  MoveL 717 to (-24.58, 53.5, 24) mm, rotated rx -180 ry 0 rz 180 deg; joints [-1.626, -7.129, -30.226, -175.862, -23.152, -3.806]
  MoveL 718 to (-28.76, 51.39, 24) mm, rotated rx 180 ry 0 rz 180 deg; joints [-1.72, -7.341, -30.414, -175.619, -23.133, -4.03]
  MoveL 719 to (-33.23, 48.62, 24) mm, rotated rx -180 ry 0 rz -180 deg; joints [-1.842, -7.567, -30.613, -175.303, -23.115, -4.321]
  MoveL 720 to (-37.7, 45.24, 24) mm, rotated rx 180 ry 0 rz 180 deg; joints [-1.991, -7.792, -30.809, -174.919, -23.098, -4.675]
  MoveL 721 to (-42.11, 41.08, 24) mm, rotated rx 180 ry 0 rz 180 deg; joints [-2.174, -8.013, -31.001, -174.448, -23.085, -5.11]
  MoveL 722 to (-46.58, 36.05, 24) mm, rotated rx -180 ry 0 rz -180 deg; joints [-2.395, -8.233, -31.193, -173.879, -23.077, -5.634]
  MoveL 723 to (-48.92, 32.78, 24) mm, rotated rx -180 ry 0 rz -180 deg; joints [-2.539, -8.348, -31.291, -173.511, -23.076, -5.974]
  MoveL 724 to (-51.1, 29.15, 24) mm, rotated rx 180 ry 0 rz 180 deg; joints [-2.698, -8.452, -31.382, -173.104, -23.079, -6.349]
  MoveL 725 to (-52.53, 26.41, 24) mm, rotated rx -180 ry 0 rz 180 deg; joints [-2.818, -8.519, -31.439, -172.797, -23.083, -6.631]
  MoveL 726 to (-54.51, 22.28, 24) mm, rotated rx 180 ry 0 rz 180 deg; joints [-2.998, -8.611, -31.519, -172.336, -23.092, -7.056]
  MoveL 727 to (-56.61, 15.99, 24) mm, rotated rx -180 ry 0 rz 180 deg; joints [-3.272, -8.702, -31.597, -171.64, -23.115, -7.697]
  MoveL 728 to (-57.94, 10.54, 24) mm, rotated rx -180 ry 0 rz 180 deg; joints [-3.509, -8.755, -31.642, -171.04, -23.14, -8.249]
  MoveL 729 to (-58.64, 4.96, 24) mm, rotated rx 180 ry 0 rz 180 deg; joints [-3.75, -8.773, -31.657, -170.433, -23.173, -8.807]
  MoveL 730 to (-58.87, 0.71, 24) mm, rotated rx 180 ry 0 rz 180 deg; joints [-3.932, -8.77, -31.655, -169.976, -23.202, -9.228]
  MoveL 731 to (-58.77, -3.71, 24) mm, rotated rx 180 ry 0 rz 180 deg; joints [-4.121, -8.748, -31.636, -169.505, -23.236, -9.661]
  MoveL 732 to (-58.13, -9.36, 24) mm, rotated rx -180 ry 0 rz -180 deg; joints [-4.361, -8.694, -31.589, -168.91, -23.285, -10.206]
  MoveL 733 to (-56.57, -16.2, 24) mm, rotated rx -180 ry 0 rz 180 deg; joints [-4.648, -8.585, -31.496, -168.205, -23.353, -10.853]
  MoveL 734 to (-54.78, -21.48, 24) mm, rotated rx -180 ry 0 rz -180 deg; joints [-4.866, -8.469, -31.397, -167.673, -23.41, -11.34]
  MoveL 735 to (-52.18, -27.29, 24) mm, rotated rx -180 ry 0 rz 180 deg; joints [-5.103, -8.309, -31.258, -167.099, -23.48, -11.864]
  MoveL 736 to (-50.38, -30.48, 24) mm, rotated rx -180 ry 0 rz 180 deg; joints [-5.232, -8.201, -31.164, -166.792, -23.521, -12.145]
  MoveL 737 to (-46.66, -35.77, 24) mm, rotated rx -180 ry 0 rz 180 deg; joints [-5.441, -7.983, -30.976, -166.296, -23.593, -12.596]
  MoveL 738 to (-43.36, -39.85, 24) mm, rotated rx -180 ry 0 rz 180 deg; joints [-5.599, -7.793, -30.81, -165.924, -23.652, -12.935]
  MoveL 739 to (-39.52, -43.58, 24) mm, rotated rx -180 ry 0 rz 180 deg; joints [-5.74, -7.577, -30.621, -165.597, -23.71, -13.232]
  MoveL 740 to (-36.23, -46.33, 24) mm, rotated rx -180 ry 0 rz -180 deg; joints [-5.842, -7.393, -30.46, -165.365, -23.755, -13.442]
  Set speed (16.7 mm/s)
  MoveL 741 to (-35.66, -46.6, 24) mm, rotated rx 180 ry 0 rz 180 deg; joints [-5.85, -7.363, -30.433, -165.347, -23.761, -13.458]
  MoveL 742 to (-35.05, -46.54, 24) mm, rotated rx -180 ry 0 rz -180 deg; joints [-5.845, -7.331, -30.405, -165.361, -23.763, -13.445]
  MoveL 743 to (-34.54, -46.18, 24) mm, rotated rx 180 ry 0 rz 180 deg; joints [-5.828, -7.307, -30.384, -165.404, -23.762, -13.405]
  MoveL 744 to (-34.69, -44.49, 24) mm, rotated rx -180 ry 0 rz 180 deg; joints [-5.758, -7.324, -30.399, -165.572, -23.744, -13.252]
  Set speed (1000.0 mm/s)
  MoveL 745 to (-26.21, -33.57, 24) mm, rotated rx -180 ry 0 rz -180 deg; joints [-5.268, -6.943, -30.062, -166.784, -23.68, -12.137]
  Set speed (5.0 mm/s)
  MoveL 746 to (-26.21, -33.57, 18) mm, rotated rx -180 ry 0 rz 180 deg; joints [-5.268, -6.879, -30.286, -166.933, -23.96, -11.975]
  MoveL 747 to (-27.9, -33.77, 18) mm, rotated rx 180 ry 0 rz 180 deg; joints [-5.283, -6.964, -30.362, -166.892, -23.954, -12.014]
  MoveL 748 to (-28.14, -34.34, 18) mm, rotated rx -180 ry 0 rz 180 deg; joints [-5.308, -6.974, -30.371, -166.831, -23.958, -12.069]
  MoveL 749 to (-28.07, -34.96, 18) mm, rotated rx 180 ry 0 rz 180 deg; joints [-5.333, -6.967, -30.365, -166.771, -23.964, -12.124]
  MoveL 750 to (-27.69, -35.46, 18) mm, rotated rx 180 ry 0 rz 180 deg; joints [-5.353, -6.946, -30.345, -166.726, -23.97, -12.165]
  Set speed (16.7 mm/s)
  MoveL 751 to (-26.15, -36.67, 18) mm, rotated rx -180 ry 0 rz -180 deg; joints [-5.397, -6.861, -30.27, -166.624, -23.989, -12.257]
  MoveL 752 to (-23.6, -38.37, 18) mm, rotated rx -180 ry 0 rz -180 deg; joints [-5.458, -6.722, -30.147, -166.486, -24.017, -12.382]
  MoveL 753 to (-18.39, -41.25, 18) mm, rotated rx 180 ry 0 rz 180 deg; joints [-5.556, -6.441, -29.896, -166.266, -24.068, -12.579]
  MoveL 754 to (-14.04, -42.78, 18) mm, rotated rx 180 ry 0 rz -180 deg; joints [-5.602, -6.212, -29.69, -166.17, -24.101, -12.665]
  MoveL 755 to (-7.62, -44.52, 18) mm, rotated rx -180 ry 0 rz -180 deg; joints [-5.647, -5.875, -29.387, -166.079, -24.143, -12.745]
  MoveL 756 to (-0.08, -45.16, 18) mm, rotated rx 180 ry 0 rz 180 deg; joints [-5.643, -5.488, -29.036, -166.108, -24.177, -12.714]
  MoveL 757 to (4.54, -44.87, 18) mm, rotated rx 180 ry 0 rz 180 deg; joints [-5.613, -5.255, -28.823, -166.192, -24.191, -12.636]
  MoveL 758 to (10.55, -43.81, 18) mm, rotated rx 180 ry 0 rz 180 deg; joints [-5.546, -4.955, -28.549, -166.365, -24.2, -12.476]
  MoveL 759 to (15.67, -42.36, 18) mm, rotated rx -180 ry 0 rz 180 deg; joints [-5.467, -4.702, -28.316, -166.562, -24.203, -12.294]
  MoveL 760 to (22.77, -38.96, 18) mm, rotated rx -180 ry 0 rz -180 deg; joints [-5.303, -4.359, -27.998, -166.966, -24.193, -11.923]
  MoveL 761 to (23.75, -38.19, 18) mm, rotated rx 180 ry 0 rz 180 deg; joints [-5.269, -4.313, -27.956, -167.05, -24.19, -11.847]
  MoveL 762 to (24.79, -37.75, 18) mm, rotated rx 180 ry 0 rz 180 deg; joints [-5.247, -4.263, -27.909, -167.103, -24.189, -11.798]
  MoveL 763 to (25.87, -36.99, 18) mm, rotated rx -180 ry 0 rz -180 deg; joints [-5.213, -4.212, -27.861, -167.187, -24.185, -11.721]
  MoveL 764 to (31.61, -32.27, 18) mm, rotated rx -180 ry 0 rz -180 deg; joints [-5.003, -3.943, -27.611, -167.697, -24.161, -11.254]
  MoveL 765 to (34.13, -29.42, 18) mm, rotated rx -180 ry 0 rz -180 deg; joints [-4.881, -3.828, -27.503, -167.994, -24.144, -10.982]
  MoveL 766 to (38.38, -23.8, 18) mm, rotated rx -180 ry 0 rz 180 deg; joints [-4.643, -3.637, -27.324, -168.572, -24.112, -10.454]
  MoveL 767 to (40.34, -20.05, 18) mm, rotated rx 180 ry 0 rz 180 deg; joints [-4.487, -3.554, -27.245, -168.948, -24.089, -10.11]
  MoveL 768 to (42.9, -14.11, 18) mm, rotated rx 180 ry 0 rz 180 deg; joints [-4.243, -3.447, -27.145, -169.54, -24.053, -9.569]
  MoveL 769 to (43.73, -10.9, 18) mm, rotated rx -180 ry 0 rz 180 deg; joints [-4.114, -3.417, -27.117, -169.855, -24.033, -9.281]
  MoveL 770 to (45.05, -3.17, 18) mm, rotated rx 180 ry 0 rz 180 deg; joints [-3.803, -3.378, -27.079, -170.611, -23.987, -8.591]
  MoveL 771 to (45.17, 0.09, 18) mm, rotated rx 180 ry 0 rz 180 deg; joints [-3.673, -3.383, -27.084, -170.927, -23.968, -8.302]
  MoveL 772 to (44.61, 6.42, 18) mm, rotated rx -180 ry 0 rz 180 deg; joints [-3.423, -3.431, -27.129, -171.536, -23.93, -7.745]
  MoveL 773 to (43.15, 13.22, 18) mm, rotated rx -180 ry 0 rz 180 deg; joints [-3.156, -3.524, -27.217, -172.188, -23.89, -7.15]
  MoveL 774 to (41.73, 17.09, 18) mm, rotated rx 180 ry 0 rz 180 deg; joints [-3.004, -3.606, -27.295, -172.557, -23.867, -6.813]
  MoveL 775 to (38.05, 24.34, 18) mm, rotated rx -180 ry 0 rz -180 deg; joints [-2.722, -3.811, -27.487, -173.248, -23.823, -6.181]
  MoveL 776 to (34.85, 28.44, 18) mm, rotated rx -180 ry 0 rz 180 deg; joints [-2.564, -3.982, -27.647, -173.635, -23.796, -5.828]
  MoveL 777 to (30.87, 32.97, 18) mm, rotated rx 180 ry 0 rz 180 deg; joints [-2.389, -4.194, -27.845, -174.064, -23.764, -5.436]
  MoveL 778 to (24.7, 37.75, 18) mm, rotated rx -180 ry 0 rz -180 deg; joints [-2.206, -4.517, -28.145, -174.51, -23.725, -5.028]
  MoveL 779 to (24.15, 37.96, 18) mm, rotated rx 180 ry 0 rz 180 deg; joints [-2.198, -4.545, -28.171, -174.528, -23.722, -5.012]
  MoveL 780 to (23.56, 38.41, 18) mm, rotated rx -180 ry 0 rz 180 deg; joints [-2.181, -4.576, -28.2, -174.571, -23.718, -4.973]
  MoveL 781 to (18.35, 41.27, 18) mm, rotated rx 180 ry 0 rz 180 deg; joints [-2.073, -4.846, -28.449, -174.834, -23.688, -4.733]
  MoveL 782 to (14.11, 42.76, 18) mm, rotated rx -180 ry 0 rz 180 deg; joints [-2.019, -5.065, -28.65, -174.965, -23.666, -4.613]
  MoveL 783 to (7.59, 44.53, 18) mm, rotated rx 180 ry 0 rz 180 deg; joints [-1.956, -5.401, -28.957, -175.116, -23.632, -4.476]
  MoveL 784 to (0.04, 45.16, 18) mm, rotated rx 180 ry 0 rz 180 deg; joints [-1.94, -5.787, -29.308, -175.148, -23.596, -4.448]
  MoveL 785 to (-5.87, 44.7, 18) mm, rotated rx 180 ry 0 rz 180 deg; joints [-1.968, -6.089, -29.58, -175.074, -23.569, -4.517]
  MoveL 786 to (-12.92, 43.24, 18) mm, rotated rx -180 ry 0 rz 180 deg; joints [-2.038, -6.448, -29.902, -174.89, -23.538, -4.687]
  MoveL 787 to (-16.08, 42.17, 18) mm, rotated rx 180 ry 0 rz 180 deg; joints [-2.087, -6.609, -30.046, -174.764, -23.525, -4.803]
  MoveL 788 to (-22.99, 38.84, 18) mm, rotated rx 180 ry 0 rz 180 deg; joints [-2.237, -6.957, -30.356, -174.382, -23.499, -5.155]
  MoveL 789 to (-23.69, 38.24, 18) mm, rotated rx 180 ry 0 rz 180 deg; joints [-2.263, -6.992, -30.387, -174.315, -23.497, -5.216]
  MoveL 790 to (-24.82, 37.73, 18) mm, rotated rx -180 ry 0 rz 180 deg; joints [-2.287, -7.049, -30.437, -174.256, -23.493, -5.271]
  MoveL 791 to (-25.9, 36.97, 18) mm, rotated rx 180 ry 0 rz 180 deg; joints [-2.32, -7.103, -30.485, -174.17, -23.49, -5.35]
  MoveL 792 to (-31.55, 32.32, 18) mm, rotated rx 180 ry 0 rz 180 deg; joints [-2.526, -7.385, -30.733, -173.649, -23.477, -5.829]
  MoveL 793 to (-34.16, 29.39, 18) mm, rotated rx 180 ry 0 rz 180 deg; joints [-2.654, -7.512, -30.845, -173.325, -23.475, -6.127]
  MoveL 794 to (-38.41, 23.76, 18) mm, rotated rx -180 ry 0 rz 180 deg; joints [-2.9, -7.718, -31.025, -172.703, -23.477, -6.698]
  MoveL 795 to (-40.36, 20, 18) mm, rotated rx -180 ry 0 rz 180 deg; joints [-3.063, -7.809, -31.104, -172.294, -23.485, -7.075]
  MoveL 796 to (-42.93, 14.05, 18) mm, rotated rx -180 ry 0 rz 180 deg; joints [-3.321, -7.924, -31.205, -171.647, -23.503, -7.669]
  MoveL 797 to (-43.76, 10.82, 18) mm, rotated rx -180 ry 0 rz -180 deg; joints [-3.46, -7.957, -31.233, -171.301, -23.518, -7.986]
  MoveL 798 to (-45.03, 3.4, 18) mm, rotated rx -180 ry 0 rz -180 deg; joints [-3.778, -7.999, -31.27, -170.511, -23.559, -8.711]
  MoveL 799 to (-45.16, 0.22, 18) mm, rotated rx -180 ry 0 rz -180 deg; joints [-3.913, -7.994, -31.266, -170.178, -23.58, -9.016]
  MoveL 800 to (-44.82, -4.92, 18) mm, rotated rx -180 ry 0 rz 180 deg; joints [-4.13, -7.958, -31.234, -169.645, -23.62, -9.504]
  MoveL 801 to (-43.65, -11.27, 18) mm, rotated rx 180 ry 0 rz 180 deg; joints [-4.395, -7.873, -31.16, -168.999, -23.676, -10.095]
  MoveL 802 to (-42.96, -13.88, 18) mm, rotated rx 180 ry 0 rz 180 deg; joints [-4.503, -7.827, -31.12, -168.737, -23.701, -10.334]
  MoveL 803 to (-41.79, -16.95, 18) mm, rotated rx -180 ry 0 rz -180 deg; joints [-4.629, -7.754, -31.056, -168.434, -23.733, -10.611]
  MoveL 804 to (-38.1, -24.27, 18) mm, rotated rx 180 ry 0 rz 180 deg; joints [-4.924, -7.532, -30.862, -167.728, -23.816, -11.255]
  MoveL 805 to (-36.06, -27.07, 18) mm, rotated rx 180 ry 0 rz 180 deg; joints [-5.034, -7.415, -30.759, -167.468, -23.851, -11.491]
  MoveL 806 to (-30.91, -32.94, 18) mm, rotated rx 180 ry 0 rz 180 deg; joints [-5.26, -7.123, -30.502, -166.939, -23.931, -11.972]
  MoveL 807 to (-27.69, -35.46, 18) mm, rotated rx 180 ry 0 rz 180 deg; joints [-5.353, -6.946, -30.345, -166.726, -23.97, -12.165]
  Set speed (16.7 mm/s)
  MoveL 808 to (-27.12, -35.7, 18) mm, rotated rx 180 ry 0 rz 180 deg; joints [-5.361, -6.915, -30.318, -166.708, -23.976, -12.181]
  MoveL 809 to (-26.51, -35.63, 18) mm, rotated rx -180 ry 0 rz -180 deg; joints [-5.355, -6.884, -30.291, -166.723, -23.978, -12.167]
  MoveL 810 to (-26.01, -35.25, 18) mm, rotated rx -180 ry 0 rz -180 deg; joints [-5.338, -6.86, -30.27, -166.767, -23.977, -12.127]
  MoveL 811 to (-26.21, -33.57, 18) mm, rotated rx 180 ry 0 rz 180 deg; joints [-5.268, -6.879, -30.286, -166.933, -23.96, -11.975]
  Set speed (1000.0 mm/s)
  MoveL 812 to (-12.43, -16.45, 18) mm, rotated rx -180 ry 0 rz 180 deg; joints [-4.51, -6.248, -29.723, -168.8, -23.88, -10.262]
  Set speed (5.0 mm/s)
  MoveL 813 to (-12.43, -16.45, 12) mm, rotated rx -180 ry 0 rz -180 deg; joints [-4.51, -6.182, -29.945, -168.925, -24.163, -10.125]
  MoveL 814 to (-14.12, -16.64, 12) mm, rotated rx 180 ry 0 rz 180 deg; joints [-4.523, -6.268, -30.022, -168.89, -24.156, -10.158]
  MoveL 815 to (-14.37, -17.21, 12) mm, rotated rx -180 ry 0 rz -180 deg; joints [-4.547, -6.278, -30.031, -168.831, -24.16, -10.212]
  MoveL 816 to (-14.3, -17.82, 12) mm, rotated rx -180 ry 0 rz -180 deg; joints [-4.572, -6.272, -30.026, -168.77, -24.165, -10.268]
  MoveL 817 to (-13.93, -18.33, 12) mm, rotated rx -180 ry 0 rz -180 deg; joints [-4.592, -6.251, -30.007, -168.724, -24.17, -10.309]
  Set speed (16.7 mm/s)
  MoveL 818 to (-13.27, -18.86, 12) mm, rotated rx 180 ry 0 rz 180 deg; joints [-4.612, -6.215, -29.975, -168.678, -24.178, -10.351]
  MoveL 819 to (-10.86, -20.34, 12) mm, rotated rx 180 ry 0 rz 180 deg; joints [-4.665, -6.086, -29.858, -168.557, -24.2, -10.461]
  MoveL 820 to (-8.3, -21.51, 12) mm, rotated rx -180 ry 0 rz -180 deg; joints [-4.705, -5.95, -29.736, -168.467, -24.22, -10.541]
  MoveL 821 to (-5.71, -22.36, 12) mm, rotated rx -180 ry 0 rz 180 deg; joints [-4.731, -5.814, -29.613, -168.411, -24.238, -10.592]
  MoveL 822 to (-2.84, -23, 12) mm, rotated rx 180 ry 0 rz 180 deg; joints [-4.747, -5.665, -29.479, -168.378, -24.255, -10.621]
  MoveL 823 to (0.04, -23.2, 12) mm, rotated rx 180 ry 0 rz 180 deg; joints [-4.745, -5.518, -29.344, -168.388, -24.268, -10.611]
  MoveL 824 to (2.55, -23.04, 12) mm, rotated rx 180 ry 0 rz 180 deg; joints [-4.73, -5.39, -29.228, -168.429, -24.276, -10.572]
  MoveL 825 to (4.71, -22.63, 12) mm, rotated rx -180 ry 0 rz 180 deg; joints [-4.707, -5.282, -29.129, -168.49, -24.281, -10.516]
  MoveL 826 to (7.7, -21.73, 12) mm, rotated rx -180 ry 0 rz 180 deg; joints [-4.66, -5.134, -28.994, -168.607, -24.285, -10.408]
  MoveL 827 to (10.34, -20.61, 12) mm, rotated rx 180 ry 0 rz 180 deg; joints [-4.606, -5.004, -28.875, -168.742, -24.286, -10.284]
  MoveL 828 to (12.82, -19.16, 12) mm, rotated rx -180 ry 0 rz 180 deg; joints [-4.539, -4.884, -28.765, -168.906, -24.283, -10.134]
  MoveL 829 to (15.05, -17.47, 12) mm, rotated rx 180 ry 0 rz 180 deg; joints [-4.463, -4.778, -28.667, -169.09, -24.278, -9.965]
  MoveL 830 to (17.03, -15.54, 12) mm, rotated rx -180 ry 0 rz 180 deg; joints [-4.379, -4.684, -28.581, -169.296, -24.271, -9.777]
  MoveL 831 to (18.85, -13.28, 12) mm, rotated rx 180 ry 0 rz 180 deg; joints [-4.282, -4.601, -28.504, -169.531, -24.261, -9.562]
  MoveL 832 to (20.34, -10.86, 12) mm, rotated rx 180 ry 0 rz 180 deg; joints [-4.18, -4.534, -28.442, -169.778, -24.249, -9.337]
  MoveL 833 to (21.5, -8.33, 12) mm, rotated rx -180 ry 0 rz -180 deg; joints [-4.074, -4.485, -28.396, -170.033, -24.236, -9.104]
  MoveL 834 to (22.34, -5.7, 12) mm, rotated rx -180 ry 0 rz -180 deg; joints [-3.966, -4.452, -28.366, -170.295, -24.221, -8.865]
  MoveL 835 to (22.85, -2.99, 12) mm, rotated rx -180 ry 0 rz -180 deg; joints [-3.855, -4.435, -28.35, -170.562, -24.206, -8.621]
  MoveL 836 to (23.04, 0.44, 12) mm, rotated rx -180 ry 0 rz 180 deg; joints [-3.716, -4.437, -28.352, -170.897, -24.185, -8.315]
  MoveL 837 to (22.58, 4.55, 12) mm, rotated rx -180 ry 0 rz -180 deg; joints [-3.551, -4.474, -28.386, -171.295, -24.159, -7.953]
  MoveL 838 to (21.92, 7.05, 12) mm, rotated rx 180 ry 0 rz 180 deg; joints [-3.452, -4.515, -28.424, -171.534, -24.143, -7.735]
  MoveL 839 to (20.59, 10.37, 12) mm, rotated rx 180 ry 0 rz 180 deg; joints [-3.321, -4.592, -28.496, -171.85, -24.12, -7.447]
  MoveL 840 to (19.25, 12.68, 12) mm, rotated rx 180 ry 0 rz -180 deg; joints [-3.231, -4.667, -28.565, -172.067, -24.102, -7.249]
  MoveL 841 to (17.5, 15.01, 12) mm, rotated rx -180 ry 0 rz -180 deg; joints [-3.14, -4.763, -28.653, -172.286, -24.084, -7.05]
  MoveL 842 to (15.49, 17.08, 12) mm, rotated rx 180 ry 0 rz 180 deg; joints [-3.061, -4.871, -28.752, -172.476, -24.066, -6.876]
  MoveL 843 to (13.35, 18.8, 12) mm, rotated rx 180 ry 0 rz 180 deg; joints [-2.995, -4.984, -28.857, -172.633, -24.049, -6.734]
  MoveL 844 to (10.93, 20.3, 12) mm, rotated rx -180 ry 0 rz -180 deg; joints [-2.939, -5.111, -28.973, -172.766, -24.032, -6.612]
  MoveL 845 to (8.27, 21.52, 12) mm, rotated rx 180 ry 0 rz 180 deg; joints [-2.895, -5.25, -29.101, -172.872, -24.015, -6.517]
  MoveL 846 to (5.67, 22.37, 12) mm, rotated rx 180 ry 0 rz 180 deg; joints [-2.866, -5.385, -29.224, -172.94, -24, -6.455]
  MoveL 847 to (2.81, 23, 12) mm, rotated rx 180 ry 0 rz 180 deg; joints [-2.846, -5.533, -29.358, -172.985, -23.985, -6.415]
  MoveL 848 to (0.03, 23.2, 12) mm, rotated rx -180 ry 0 rz 180 deg; joints [-2.843, -5.675, -29.488, -172.987, -23.972, -6.413]
  MoveL 849 to (-2.49, 23.04, 12) mm, rotated rx 180 ry 0 rz 180 deg; joints [-2.855, -5.803, -29.604, -172.956, -23.961, -6.443]
  MoveL 850 to (-4.65, 22.65, 12) mm, rotated rx -180 ry 0 rz 180 deg; joints [-2.876, -5.913, -29.703, -172.902, -23.953, -6.492]
  MoveL 851 to (-7.73, 21.72, 12) mm, rotated rx -180 ry 0 rz 180 deg; joints [-2.92, -6.069, -29.843, -172.789, -23.943, -6.597]
  MoveL 852 to (-10.37, 20.59, 12) mm, rotated rx -180 ry 0 rz -180 deg; joints [-2.972, -6.201, -29.962, -172.657, -23.936, -6.718]
  MoveL 853 to (-12.76, 19.2, 12) mm, rotated rx 180 ry 0 rz 180 deg; joints [-3.035, -6.32, -30.068, -172.5, -23.931, -6.862]
  MoveL 854 to (-14.99, 17.52, 12) mm, rotated rx -180 ry 0 rz -180 deg; joints [-3.11, -6.429, -30.167, -172.313, -23.929, -7.034]
  MoveL 855 to (-17.06, 15.51, 12) mm, rotated rx 180 ry 0 rz 180 deg; joints [-3.198, -6.53, -30.257, -172.094, -23.929, -7.234]
  MoveL 856 to (-18.8, 13.35, 12) mm, rotated rx 180 ry 0 rz 180 deg; joints [-3.292, -6.613, -30.331, -171.861, -23.932, -7.447]
  MoveL 857 to (-20.29, 10.95, 12) mm, rotated rx 180 ry 0 rz 180 deg; joints [-3.396, -6.682, -30.392, -171.606, -23.938, -7.681]
  MoveL 858 to (-21.52, 8.27, 12) mm, rotated rx 180 ry 0 rz 180 deg; joints [-3.51, -6.737, -30.441, -171.324, -23.948, -7.939]
  MoveL 859 to (-22.36, 5.63, 12) mm, rotated rx -180 ry 0 rz -180 deg; joints [-3.622, -6.772, -30.472, -171.049, -23.96, -8.19]
  MoveL 860 to (-22.87, 2.9, 12) mm, rotated rx 180 ry 0 rz 180 deg; joints [-3.738, -6.789, -30.487, -170.767, -23.975, -8.448]
  MoveL 861 to (-23.06, 0.04, 12) mm, rotated rx -180 ry 0 rz 180 deg; joints [-3.858, -6.789, -30.487, -170.476, -23.992, -8.714]
  MoveL 862 to (-22.93, -2.29, 12) mm, rotated rx -180 ry 0 rz 180 deg; joints [-3.954, -6.774, -30.474, -170.242, -24.009, -8.928]
  MoveL 863 to (-22.29, -5.75, 12) mm, rotated rx 180 ry 0 rz 180 deg; joints [-4.097, -6.729, -30.434, -169.899, -24.036, -9.241]
  MoveL 864 to (-21.73, -7.73, 12) mm, rotated rx -180 ry 0 rz -180 deg; joints [-4.177, -6.693, -30.402, -169.705, -24.053, -9.418]
  MoveL 865 to (-20.65, -10.24, 12) mm, rotated rx 180 ry 0 rz 180 deg; joints [-4.279, -6.628, -30.344, -169.463, -24.077, -9.638]
  MoveL 866 to (-19.16, -12.83, 12) mm, rotated rx 180 ry 0 rz 180 deg; joints [-4.381, -6.541, -30.267, -169.219, -24.104, -9.86]
  MoveL 867 to (-17.55, -14.95, 12) mm, rotated rx 180 ry 0 rz 180 deg; joints [-4.464, -6.45, -30.185, -169.023, -24.127, -10.038]
  MoveL 868 to (-15.54, -17.04, 12) mm, rotated rx -180 ry 0 rz -180 deg; joints [-4.544, -6.339, -30.086, -168.836, -24.153, -10.208]
  MoveL 869 to (-13.93, -18.33, 12) mm, rotated rx -180 ry 0 rz -180 deg; joints [-4.592, -6.251, -30.007, -168.724, -24.17, -10.309]
  Set speed (16.7 mm/s)
  MoveL 870 to (-13.36, -18.58, 12) mm, rotated rx -180 ry 0 rz -180 deg; joints [-4.6, -6.221, -29.98, -168.705, -24.175, -10.326]
  MoveL 871 to (-12.75, -18.51, 12) mm, rotated rx 180 ry 0 rz 180 deg; joints [-4.596, -6.19, -29.952, -168.718, -24.177, -10.314]
  MoveL 872 to (-12.24, -18.14, 12) mm, rotated rx -180 ry 0 rz -180 deg; joints [-4.579, -6.166, -29.93, -168.76, -24.177, -10.276]
  MoveL 873 to (-12.43, -16.45, 12) mm, rotated rx -180 ry 0 rz 180 deg; joints [-4.51, -6.182, -29.945, -168.925, -24.163, -10.125]
  MoveL 874 to (-12.43, -16.45, 13.2) mm, rotated rx 180 ry 0 rz 180 deg; joints [-4.51, -6.195, -29.901, -168.901, -24.106, -10.152]
  Set speed (1000.0 mm/s)
  MoveL 875 to (-12.43, -16.45, 61) mm, rotated rx 180 ry 0 rz 180 deg; joints [-4.51, -6.673, -28.096, -167.815, -21.871, -11.331]
  Set speed (1000.0 mm/s)
  MoveL 876 to (-12.43, -16.45, 61) mm, rotated rx 180 ry 0 rz 180 deg; joints [-4.51, -6.673, -28.096, -167.815, -21.871, -11.331]
  MoveL 877 to (-12.43, -16.45, 161) mm, rotated rx -180 ry 0 rz -180 deg; joints [-4.51, -7.348, -24.071, -164.672, -17.303, -14.665]
